SUBAPPLICATION mapping_Softkeys_IE (* Mapping for all Softkey *)
  (* Standard: 61499-2 *)
  (* Version 1.0, 2023-01-29, Franz *)
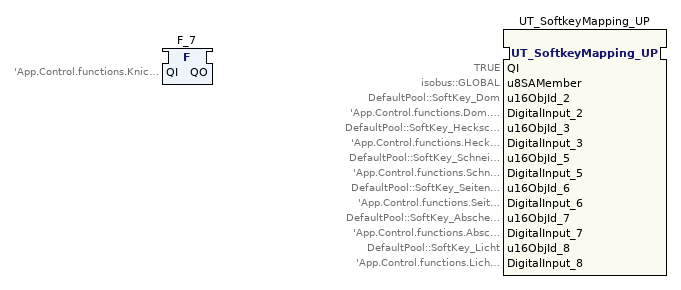
  FBS
    UT_SoftkeyMapping_UP : UT_SoftkeyMapping_UP(QI := TRUE, u8SAMember := isobus::GLOBAL, u16ObjId_2 := DefaultPool::SoftKey_Dom, DigitalInput_2 := 'App.Control.functions.Dom.SoftKey', u16ObjId_3 := DefaultPool::SoftKey_Heckschieber, DigitalInput_3 := 'App.Control.functions.Heckschieber.SoftKey', u16ObjId_5 := DefaultPool::SoftKey_Schneidwerk, DigitalInput_5 := 'App.Control.functions.Schneidwerk.SoftKey', u16ObjId_6 := DefaultPool::SoftKey_Seitenschieber, DigitalInput_6 := 'App.Control.functions.Seitenschieber.SoftKey', u16ObjId_7 := DefaultPool::SoftKey_Abscheider, DigitalInput_7 := 'App.Control.functions.Abscheider.SoftKey', u16ObjId_8 := DefaultPool::SoftKey_Licht, DigitalInput_8 := 'App.Control.functions.Licht.SoftKey');
  END_FBS
  SUBAPPS
    F_7 : F(QI := 'App.Control.functions.Knickdeichsel.SoftKey_heben.IX');
  END_SUBAPPS
END_SUBAPPLICATION
